TYPE (* One recipe step as a struct: StepType/CmdTargetName/CmdStateArr/Wait1Id/Wait1State/NextStep/AltCount/TermCount *)
  (* Standard: 1131-3 *)
  (* Version 0.1, 5/24/2026, easensoy, WMG, array-of-struct packaging of the 6 recipe arrays *)
  PACKAGE Main;
  RecipeStep : STRUCT
    StepType : INT;
    CmdTargetName : STRING[150];
    CmdStateArr : INT;
    Wait1Id : INT;
    Wait1State : INT;
    NextStep : INT;
    AltCount : INT;
    TermCount : INT;
  END_STRUCT;
END_TYPE
(* other elements stored in the file *)
(* A WAIT is a sum of products: AltCount alternatives from this row, each of TermCount rows that hold together. It releases when ANY alternative holds. Zero reads as one alternative of one term, which is the plain single-slot wait. *)
